FUNCTION_BLOCK X2Y2S_ST (* Compute X^2-Y^2(scanned, ST language) *)
  (* Standard: 61499-1 *)
  (* Version 0.0, 2003-08-17, JHC, Rockwell Automation, Adapted from X2Y2S. *)
  (* Compiler header: package fb.rt.student; *)
  (* Compiler Java IBM Jikes 1.0.6 *)
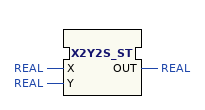
  VAR_INPUT
    X : REAL;
    Y : REAL;
  END_VAR
  VAR_OUTPUT
    OUT : REAL;
  END_VAR
  ALGORITHM REQ IN ST: (* Normally executed algorithm *)
OUT := (X-Y)*(X+Y);
  END_ALGORITHM
END_FUNCTION_BLOCK
